(* IEC 61131-3 sources: PLC-AI-Fault-Analyzer/CODESYS, 5 files *)

(* ---- codesys_constants.st ---- *)
{attribute 'qualified_only'}
VAR_GLOBAL CONSTANT
    MODE_IDLE : UINT := 0;
    MODE_CONVEYOR : UINT := 10;
    MODE_TRAFFIC_CONTROL : UINT := 20;
    MODE_PUMP_STATION : UINT := 30;
    MODE_ELEVATOR : UINT := 40;
    MODE_TUNNEL_VENTILATION : UINT := 50;
    MODE_GARAGE_DOOR : UINT := 60;

    FAULT_NONE : UINT := 0;
    FAULT_TRAFFIC_PHASE_CONFLICT : UINT := 101;
    FAULT_PUMP_STATION_FAILURE : UINT := 201;
    FAULT_ELEVATOR_DOOR_TIMEOUT : UINT := 301;
    FAULT_TUNNEL_VENTILATION_FAILURE : UINT := 401;
    FAULT_GARAGE_DOOR_SAFETY_LOCKOUT : UINT := 501;
    FAULT_CONVEYOR_JAM : UINT := 601;
END_VAR

(* ---- codesys_globals.st ---- *)
{attribute 'qualified_only'}
VAR_GLOBAL
    Conveyor_Running : BOOL := FALSE;
    Sensor_Blocked : BOOL := FALSE;
    Motor_Current : UINT := 18;
    Safety_OK : BOOL := TRUE;
    Start_Command : BOOL := FALSE;
    Stop_Command : BOOL := FALSE;
    Reset_Command : BOOL := FALSE;
    Tank_Level_Low : BOOL := FALSE;
    Tank_Level_High : BOOL := TRUE;
    Sequence_Timeout : BOOL := FALSE;
    System_Fault_Latch : BOOL := FALSE;
    Pump_Running : BOOL := FALSE;
    HVAC_Fault : BOOL := FALSE;
    Mode_Code : UINT := GVL_Constants.MODE_IDLE;
    Fault_Code : UINT := GVL_Constants.FAULT_NONE;

    HoldingRegs : ARRAY[0..14] OF UINT;
END_VAR

(* ---- codesys_scenario_globals.st ---- *)
{attribute 'qualified_only'}
VAR_GLOBAL
    ScenarioName : STRING[40] := 'idle';
    LoadScenario : BOOL := TRUE;
    ScenarioLoaded : BOOL := FALSE;
    LastLoadedScenario : STRING[40] := '';
END_VAR

(* ---- codesys_fb_scenario_demo_loader.st ---- *)
FUNCTION_BLOCK FB_ScenarioDemoLoader
VAR_INPUT
    Execute : BOOL;
    ScenarioName : STRING[40];
END_VAR
VAR_OUTPUT
    Done : BOOL;
    ActiveScenario : STRING[40];
END_VAR
VAR
    PreviousExecute : BOOL;
    RisingEdge : BOOL;
END_VAR

RisingEdge := Execute AND NOT PreviousExecute;
PreviousExecute := Execute;

IF RisingEdge THEN
    GVL_Diagnostics.Conveyor_Running := FALSE;
    GVL_Diagnostics.Sensor_Blocked := FALSE;
    GVL_Diagnostics.Motor_Current := 18;
    GVL_Diagnostics.Safety_OK := TRUE;
    GVL_Diagnostics.Start_Command := FALSE;
    GVL_Diagnostics.Stop_Command := FALSE;
    GVL_Diagnostics.Reset_Command := FALSE;
    GVL_Diagnostics.Tank_Level_Low := FALSE;
    GVL_Diagnostics.Tank_Level_High := TRUE;
    GVL_Diagnostics.Sequence_Timeout := FALSE;
    GVL_Diagnostics.System_Fault_Latch := FALSE;
    GVL_Diagnostics.Pump_Running := FALSE;
    GVL_Diagnostics.HVAC_Fault := FALSE;
    GVL_Diagnostics.Mode_Code := GVL_Constants.MODE_IDLE;
    GVL_Diagnostics.Fault_Code := GVL_Constants.FAULT_NONE;

    IF ScenarioName = 'traffic_phase_conflict' THEN
        GVL_Diagnostics.Start_Command := TRUE;
        GVL_Diagnostics.Stop_Command := TRUE;
        GVL_Diagnostics.System_Fault_Latch := TRUE;
        GVL_Diagnostics.Mode_Code := GVL_Constants.MODE_TRAFFIC_CONTROL;
        GVL_Diagnostics.Fault_Code := GVL_Constants.FAULT_TRAFFIC_PHASE_CONFLICT;

    ELSIF ScenarioName = 'pump_station_failure' THEN
        GVL_Diagnostics.Start_Command := TRUE;
        GVL_Diagnostics.Tank_Level_Low := TRUE;
        GVL_Diagnostics.Tank_Level_High := TRUE;
        GVL_Diagnostics.Sequence_Timeout := TRUE;
        GVL_Diagnostics.System_Fault_Latch := TRUE;
        GVL_Diagnostics.Pump_Running := TRUE;
        GVL_Diagnostics.Mode_Code := GVL_Constants.MODE_PUMP_STATION;
        GVL_Diagnostics.Fault_Code := GVL_Constants.FAULT_PUMP_STATION_FAILURE;

    ELSIF ScenarioName = 'elevator_door_fault' THEN
        GVL_Diagnostics.Sensor_Blocked := TRUE;
        GVL_Diagnostics.Safety_OK := FALSE;
        GVL_Diagnostics.Start_Command := TRUE;
        GVL_Diagnostics.Sequence_Timeout := TRUE;
        GVL_Diagnostics.System_Fault_Latch := TRUE;
        GVL_Diagnostics.Mode_Code := GVL_Constants.MODE_ELEVATOR;
        GVL_Diagnostics.Fault_Code := GVL_Constants.FAULT_ELEVATOR_DOOR_TIMEOUT;

    ELSIF ScenarioName = 'tunnel_ventilation_fault' THEN
        GVL_Diagnostics.Start_Command := TRUE;
        GVL_Diagnostics.Sequence_Timeout := TRUE;
        GVL_Diagnostics.System_Fault_Latch := TRUE;
        GVL_Diagnostics.HVAC_Fault := TRUE;
        GVL_Diagnostics.Mode_Code := GVL_Constants.MODE_TUNNEL_VENTILATION;
        GVL_Diagnostics.Fault_Code := GVL_Constants.FAULT_TUNNEL_VENTILATION_FAILURE;

    ELSIF ScenarioName = 'garage_door_fault' THEN
        GVL_Diagnostics.Sensor_Blocked := TRUE;
        GVL_Diagnostics.Safety_OK := FALSE;
        GVL_Diagnostics.Start_Command := TRUE;
        GVL_Diagnostics.Sequence_Timeout := TRUE;
        GVL_Diagnostics.System_Fault_Latch := TRUE;
        GVL_Diagnostics.Mode_Code := GVL_Constants.MODE_GARAGE_DOOR;
        GVL_Diagnostics.Fault_Code := GVL_Constants.FAULT_GARAGE_DOOR_SAFETY_LOCKOUT;

    ELSIF ScenarioName = 'conveyor_jam' THEN
        GVL_Diagnostics.Conveyor_Running := TRUE;
        GVL_Diagnostics.Sensor_Blocked := TRUE;
        GVL_Diagnostics.Motor_Current := 95;
        GVL_Diagnostics.Start_Command := TRUE;
        GVL_Diagnostics.Sequence_Timeout := TRUE;
        GVL_Diagnostics.System_Fault_Latch := TRUE;
        GVL_Diagnostics.Mode_Code := GVL_Constants.MODE_CONVEYOR;
        GVL_Diagnostics.Fault_Code := GVL_Constants.FAULT_CONVEYOR_JAM;

    ELSE
        GVL_Diagnostics.Mode_Code := GVL_Constants.MODE_IDLE;
        GVL_Diagnostics.Fault_Code := GVL_Constants.FAULT_NONE;
    END_IF

    ActiveScenario := ScenarioName;
    Done := TRUE;
ELSE
    Done := FALSE;
END_IF

(* ---- codesys_main.st ---- *)
PROGRAM PLC_PRG
VAR
    ScenarioLoader : FB_ScenarioDemoLoader;
END_VAR

ScenarioLoader(
    Execute := GVL_Scenario.LoadScenario,
    ScenarioName := GVL_Scenario.ScenarioName
);

IF ScenarioLoader.Done THEN
    GVL_Scenario.ScenarioLoaded := TRUE;
    GVL_Scenario.LastLoadedScenario := ScenarioLoader.ActiveScenario;
    GVL_Scenario.LoadScenario := FALSE;
END_IF

IF GVL_Diagnostics.Reset_Command THEN
    GVL_Diagnostics.System_Fault_Latch := FALSE;
    GVL_Diagnostics.Sequence_Timeout := FALSE;
    GVL_Diagnostics.HVAC_Fault := FALSE;
    GVL_Diagnostics.Fault_Code := GVL_Constants.FAULT_NONE;
    GVL_Diagnostics.Reset_Command := FALSE;
END_IF

IF (GVL_Diagnostics.Fault_Code <> GVL_Constants.FAULT_NONE) THEN
    GVL_Diagnostics.System_Fault_Latch := TRUE;
END_IF

(* Modbus TCP holding register mapping for portfolio clarity.
   Configure the CODESYS Modbus TCP server so GVL_Diagnostics.HoldingRegs[0..14]
   are exposed as holding registers 0 through 14.

   Register 0  -> Conveyor_Running
   Register 1  -> Sensor_Blocked
   Register 2  -> Motor_Current
   Register 3  -> Safety_OK
   Register 4  -> Start_Command
   Register 5  -> Stop_Command
   Register 6  -> Reset_Command
   Register 7  -> Tank_Level_Low
   Register 8  -> Tank_Level_High
   Register 9  -> Sequence_Timeout
   Register 10 -> System_Fault_Latch
   Register 11 -> Pump_Running
   Register 12 -> HVAC_Fault
   Register 13 -> Mode_Code
   Register 14 -> Fault_Code
*)
GVL_Diagnostics.HoldingRegs[0] := BOOL_TO_UINT(GVL_Diagnostics.Conveyor_Running);
GVL_Diagnostics.HoldingRegs[1] := BOOL_TO_UINT(GVL_Diagnostics.Sensor_Blocked);
GVL_Diagnostics.HoldingRegs[2] := GVL_Diagnostics.Motor_Current;
GVL_Diagnostics.HoldingRegs[3] := BOOL_TO_UINT(GVL_Diagnostics.Safety_OK);
GVL_Diagnostics.HoldingRegs[4] := BOOL_TO_UINT(GVL_Diagnostics.Start_Command);
GVL_Diagnostics.HoldingRegs[5] := BOOL_TO_UINT(GVL_Diagnostics.Stop_Command);
GVL_Diagnostics.HoldingRegs[6] := BOOL_TO_UINT(GVL_Diagnostics.Reset_Command);
GVL_Diagnostics.HoldingRegs[7] := BOOL_TO_UINT(GVL_Diagnostics.Tank_Level_Low);
GVL_Diagnostics.HoldingRegs[8] := BOOL_TO_UINT(GVL_Diagnostics.Tank_Level_High);
GVL_Diagnostics.HoldingRegs[9] := BOOL_TO_UINT(GVL_Diagnostics.Sequence_Timeout);
GVL_Diagnostics.HoldingRegs[10] := BOOL_TO_UINT(GVL_Diagnostics.System_Fault_Latch);
GVL_Diagnostics.HoldingRegs[11] := BOOL_TO_UINT(GVL_Diagnostics.Pump_Running);
GVL_Diagnostics.HoldingRegs[12] := BOOL_TO_UINT(GVL_Diagnostics.HVAC_Fault);
GVL_Diagnostics.HoldingRegs[13] := GVL_Diagnostics.Mode_Code;
GVL_Diagnostics.HoldingRegs[14] := GVL_Diagnostics.Fault_Code;
